FUNCTION Convert_DWORD_TO_DWORD : BOOL
VAR_INPUT
	in : DWORD;
	out : REFERENCE TO DWORD;
END_VAR

out := in;
Convert_DWORD_TO_DWORD := TRUE;

END_FUNCTION

(* stored: Version 1.1.0.1, ProductVersion 3.1.4024.12
   POU Convert_DWORD_TO_DWORD: Id {f4a345bd-bb9f-4f6d-b0c7-35b7c73b976f}, SpecialFunc None *)
